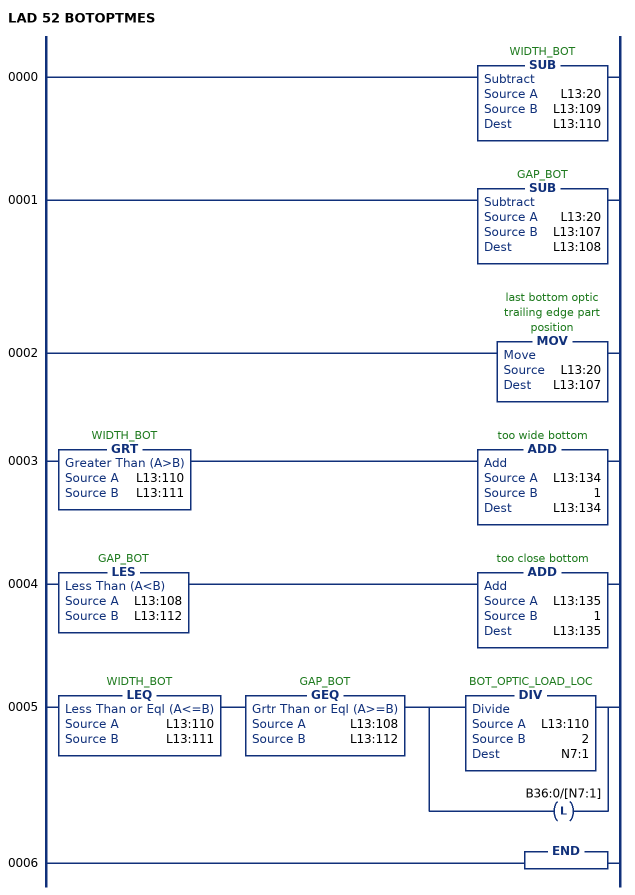
% Rung: 0 %
SOR SUB L13:20 L13:109 L13:110 EOR
%   L13:20  BOT_POSITION %
%   L13:109  BOT_LEAD_EDGE  "last bottom optic leading edge position" %
%   L13:110  WIDTH_BOT %
% Rung: 1 %
SOR SUB L13:20 L13:107 L13:108 EOR
%   L13:20  BOT_POSITION %
%   L13:107  "last bottom optic trailing edge part position" %
%   L13:108  GAP_BOT %
% Rung: 2 %
SOR MOV L13:20 L13:107 EOR
%   L13:20  BOT_POSITION %
%   L13:107  "last bottom optic trailing edge part position" %
% Rung: 3 %
SOR GRT L13:110 L13:111 ADD L13:134 1 L13:134 EOR
%   L13:110  WIDTH_BOT %
%   L13:111  BOT_MAX_WIDTH %
%   L13:134  "too wide bottom" %
% Rung: 4 %
SOR LES L13:108 L13:112 ADD L13:135 1 L13:135 EOR
%   L13:108  GAP_BOT %
%   L13:112  BOT_MIN_GAP %
%   L13:135  "too close bottom" %
% Rung: 5 %
SOR LEQ L13:110 L13:111 GEQ L13:108 L13:112 BST DIV L13:110 2 N7:1 NXB OTL B36:0/[N7:1] BND EOR
%   L13:110  WIDTH_BOT %
%   L13:111  BOT_MAX_WIDTH %
%   L13:108  GAP_BOT %
%   L13:112  BOT_MIN_GAP %
%   N7:1  BOT_OPTIC_LOAD_LOC %
%   B36:0  BOT_GOOD %
% Rung: 6 %
SOR END EOR

LADDER 60 "1 INS1"
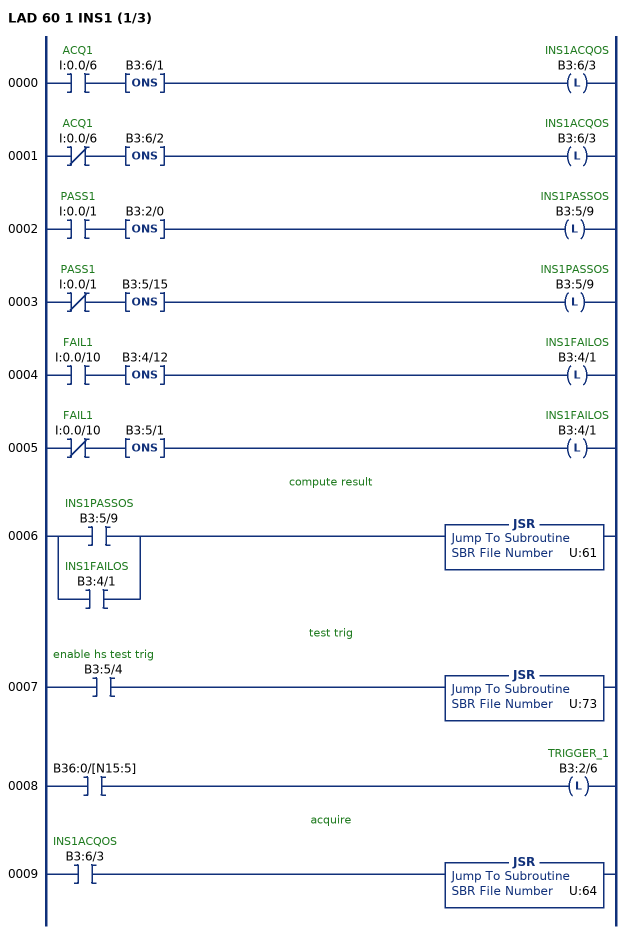
% Rung: 0 %
SOR XIC I:0.0/6 ONS B3:6/1 OTL B3:6/3 EOR
%   I:0.0/6  ACQ1 %
%   B3:6/3  INS1ACQOS %
% Rung: 1 %
SOR XIO I:0.0/6 ONS B3:6/2 OTL B3:6/3 EOR
%   I:0.0/6  ACQ1 %
%   B3:6/3  INS1ACQOS %
% Rung: 2 %
SOR XIC I:0.0/1 ONS B3:2/0 OTL B3:5/9 EOR
%   I:0.0/1  PASS1 %
%   B3:5/9  INS1PASSOS %
% Rung: 3 %
SOR XIO I:0.0/1 ONS B3:5/15 OTL B3:5/9 EOR
%   I:0.0/1  PASS1 %
%   B3:5/9  INS1PASSOS %
% Rung: 4 %
SOR XIC I:0.0/10 ONS B3:4/12 OTL B3:4/1 EOR
%   I:0.0/10  FAIL1 %
%   B3:4/1  INS1FAILOS %
% Rung: 5 %
SOR XIO I:0.0/10 ONS B3:5/1 OTL B3:4/1 EOR
%   I:0.0/10  FAIL1 %
%   B3:4/1  INS1FAILOS %
% Rung: 6 %
% compute result %
SOR BST XIC B3:5/9 NXB XIC B3:4/1 BND JSR U:61 EOR
%   B3:5/9  INS1PASSOS %
%   B3:4/1  INS1FAILOS %
% Rung: 7 %
% test trig %
SOR XIC B3:5/4 JSR U:73 EOR
%   B3:5/4  "enable hs test trig" %
% Rung: 8 %
SOR XIC B36:0/[N15:5] OTL B3:2/6 EOR
%   B36:0  BOT_GOOD %
%   N15:5  INS_1_TRIG_LOC %
%   B3:2/6  TRIGGER_1 %
% Rung: 9 %
% acquire %
SOR XIC B3:6/3 JSR U:64 EOR
%   B3:6/3  INS1ACQOS %

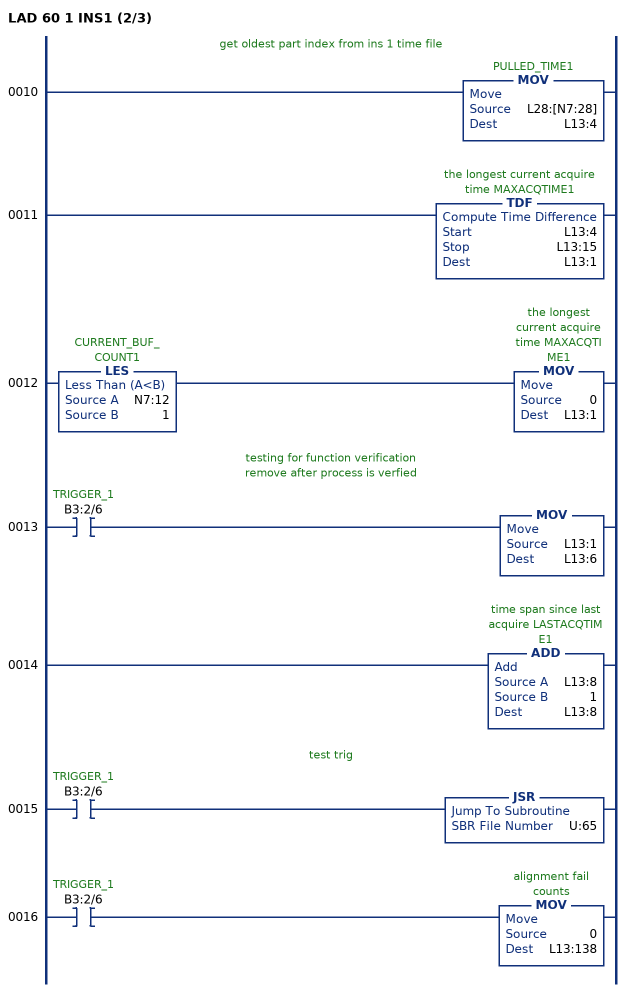
% Rung: 10 %
% get oldest part index from ins 1 time file %
SOR MOV L28:[N7:28] L13:4 EOR
%   N7:28  OLDEST_PART_INDEX1 %
%   L13:4  PULLED_TIME1 %
% Rung: 11 %
SOR TDF L13:4 L13:15 L13:1 EOR
%   L13:4  PULLED_TIME1 %
%   L13:15  THE_TIME %
%   L13:1  MAXACQTIME1  "the longest current acquire time" %
% Rung: 12 %
SOR LES N7:12 1 MOV 0 L13:1 EOR
%   N7:12  CURRENT_BUF_COUNT1 %
%   L13:1  MAXACQTIME1  "the longest current acquire time" %
% Rung: 13 %
% testing for function verification
% remove after process is verfied %
SOR XIC B3:2/6 MOV L13:1 L13:6 EOR
%   B3:2/6  TRIGGER_1 %
%   L13:1  MAXACQTIME1  "the longest current acquire time" %
% Rung: 14 %
SOR ADD L13:8 1 L13:8 EOR
%   L13:8  LASTACQTIME1  "time span since last acquire" %
% Rung: 15 %
% test trig %
SOR XIC B3:2/6 JSR U:65 EOR
%   B3:2/6  TRIGGER_1 %
% Rung: 16 %
SOR XIC B3:2/6 MOV 0 L13:138 EOR
%   B3:2/6  TRIGGER_1 %
%   L13:138  "alignment fail counts" %

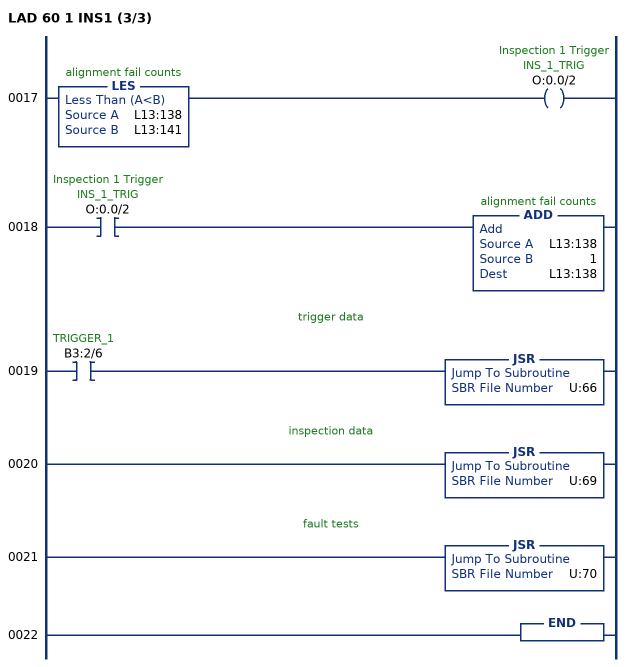
% Rung: 17 %
SOR LES L13:138 L13:141 OTE O:0.0/2 EOR
%   L13:138  "alignment fail counts" %
%   O:0.0/2  INS_1_TRIG  "Inspection 1 Trigger" %
% Rung: 18 %
SOR XIC O:0.0/2 ADD L13:138 1 L13:138 EOR
%   O:0.0/2  INS_1_TRIG  "Inspection 1 Trigger" %
%   L13:138  "alignment fail counts" %
% Rung: 19 %
% trigger data %
SOR XIC B3:2/6 JSR U:66 EOR
%   B3:2/6  TRIGGER_1 %
% Rung: 20 %
% inspection data %
SOR JSR U:69 EOR
% Rung: 21 %
% fault tests %
SOR JSR U:70 EOR
% Rung: 22 %
SOR END EOR

LADDER 61 "2 INS1RESU"
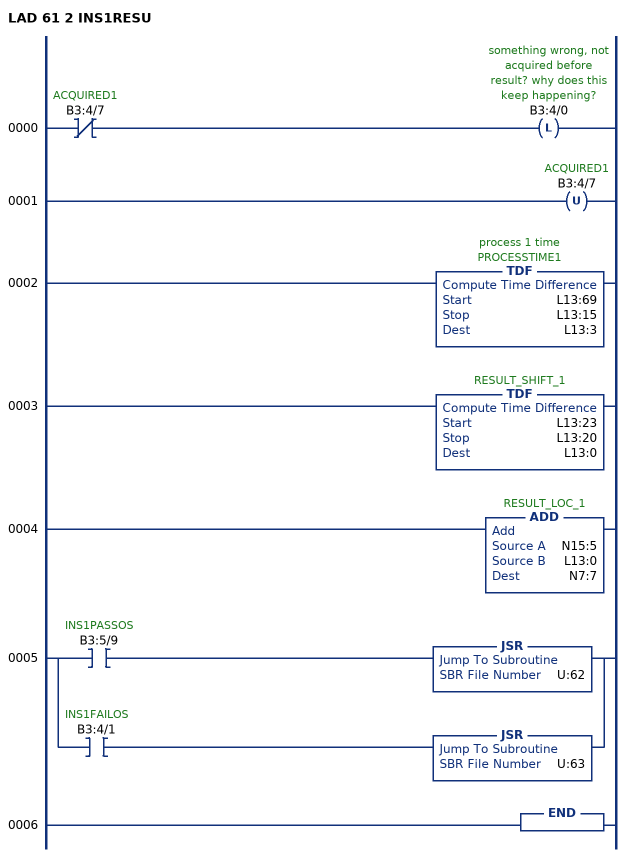
% Rung: 0 %
SOR XIO B3:4/7 OTL B3:4/0 EOR
%   B3:4/7  ACQUIRED1 %
%   B3:4/0  "something wrong, not acquired before result? why does this keep happening?" %
% Rung: 1 %
SOR OTU B3:4/7 EOR
%   B3:4/7  ACQUIRED1 %
% Rung: 2 %
SOR TDF L13:69 L13:15 L13:3 EOR
%   L13:69  TIMEOFACQ1  "the time of the last acquire" %
%   L13:15  THE_TIME %
%   L13:3  PROCESSTIME1  "process 1 time" %
% Rung: 3 %
SOR TDF L13:23 L13:20 L13:0 EOR
%   L13:23  PROCESS_START_POS_1 %
%   L13:20  BOT_POSITION %
%   L13:0  RESULT_SHIFT_1 %
% Rung: 4 %
SOR ADD N15:5 L13:0 N7:7 EOR
%   N15:5  INS_1_TRIG_LOC %
%   L13:0  RESULT_SHIFT_1 %
%   N7:7  RESULT_LOC_1 %
% Rung: 5 %
SOR BST XIC B3:5/9 JSR U:62 NXB XIC B3:4/1 JSR U:63 BND EOR
%   B3:5/9  INS1PASSOS %
%   B3:4/1  INS1FAILOS %
% Rung: 6 %
SOR END EOR

LADDER 62 "3 INS1PASS"
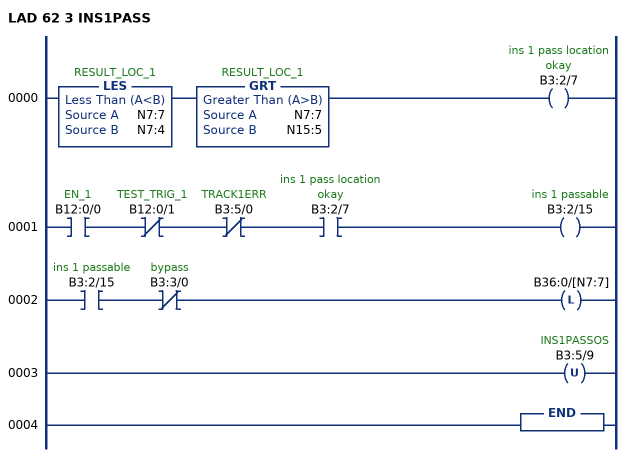
% Rung: 0 %
SOR LES N7:7 N7:4 GRT N7:7 N15:5 OTE B3:2/7 EOR
%   N7:7  RESULT_LOC_1 %
%   N7:4  INS1_MAX_SHIFT  "ins 1 maximum result location" %
%   N15:5  INS_1_TRIG_LOC %
%   B3:2/7  "ins 1 pass location okay" %
% Rung: 1 %
SOR XIC B12:0/0 XIO B12:0/1 XIO B3:5/0 XIC B3:2/7 OTE B3:2/15 EOR
%   B12:0/0  EN_1 %
%   B12:0/1  TEST_TRIG_1 %
%   B3:5/0  TRACK1ERR %
%   B3:2/7  "ins 1 pass location okay" %
%   B3:2/15  "ins 1 passable" %
% Rung: 2 %
SOR XIC B3:2/15 XIO B3:3/0 OTL B36:0/[N7:7] EOR
%   B3:2/15  "ins 1 passable" %
%   B3:3/0  "bypass" %
%   B36:0  BOT_GOOD %
%   N7:7  RESULT_LOC_1 %
% Rung: 3 %
SOR OTU B3:5/9 EOR
%   B3:5/9  INS1PASSOS %
% Rung: 4 %
SOR END EOR

LADDER 63 "4 INS1FAIL"
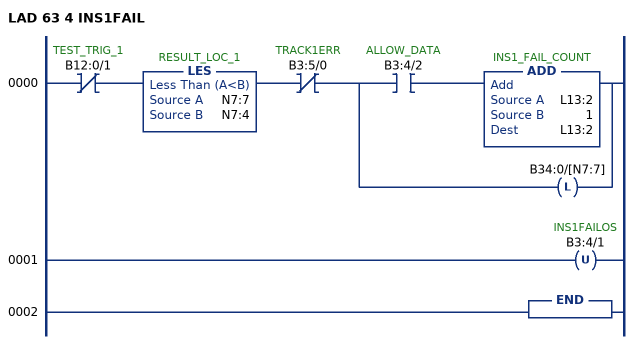
% Rung: 0 %
SOR XIO B12:0/1 LES N7:7 N7:4 XIO B3:5/0 BST XIC B3:4/2 ADD L13:2 1 L13:2 NXB OTL B34:0/[N7:7] BND EOR
%   B12:0/1  TEST_TRIG_1 %
%   N7:7  RESULT_LOC_1 %
%   N7:4  INS1_MAX_SHIFT  "ins 1 maximum result location" %
%   B3:5/0  TRACK1ERR %
%   B3:4/2  ALLOW_DATA %
%   L13:2  INS1_FAIL_COUNT %
%   B34:0  BOT_NG %
% Rung: 1 %
SOR OTU B3:4/1 EOR
%   B3:4/1  INS1FAILOS %
% Rung: 2 %
SOR END EOR

LADDER 64 "5 INS1ACQ"
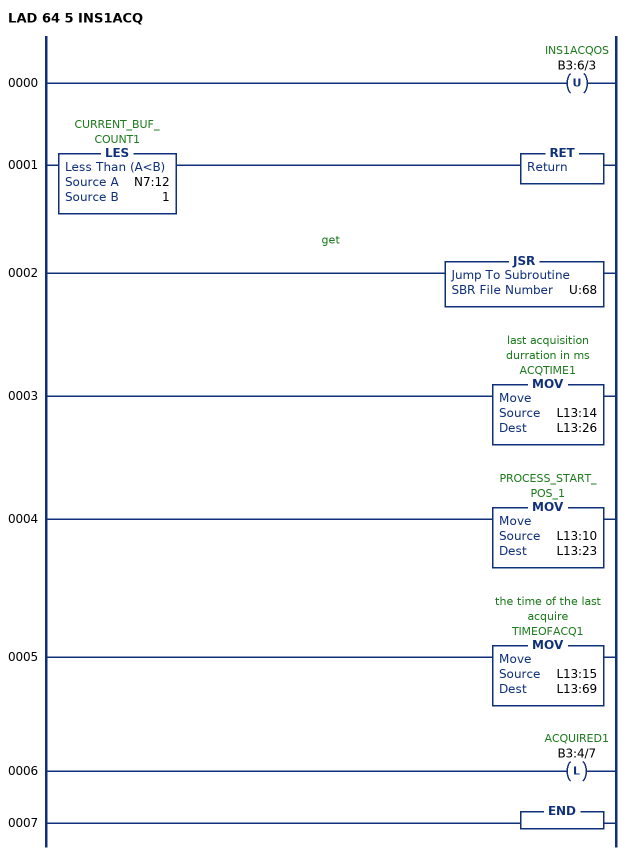
% Rung: 0 %
SOR OTU B3:6/3 EOR
%   B3:6/3  INS1ACQOS %
% Rung: 1 %
SOR LES N7:12 1 RET EOR
%   N7:12  CURRENT_BUF_COUNT1 %
% Rung: 2 %
% get %
SOR JSR U:68 EOR
% Rung: 3 %
SOR MOV L13:14 L13:26 EOR
%   L13:14  TIME_SPAN1 %
%   L13:26  ACQTIME1  "last acquisition durration in ms" %
% Rung: 4 %
SOR MOV L13:10 L13:23 EOR
%   L13:10  PULLED_POSITION1 %
%   L13:23  PROCESS_START_POS_1 %
% Rung: 5 %
SOR MOV L13:15 L13:69 EOR
%   L13:15  THE_TIME %
%   L13:69  TIMEOFACQ1  "the time of the last acquire" %
% Rung: 6 %
SOR OTL B3:4/7 EOR
%   B3:4/7  ACQUIRED1 %
% Rung: 7 %
SOR END EOR

LADDER 65 "6 Q1TESTTR"
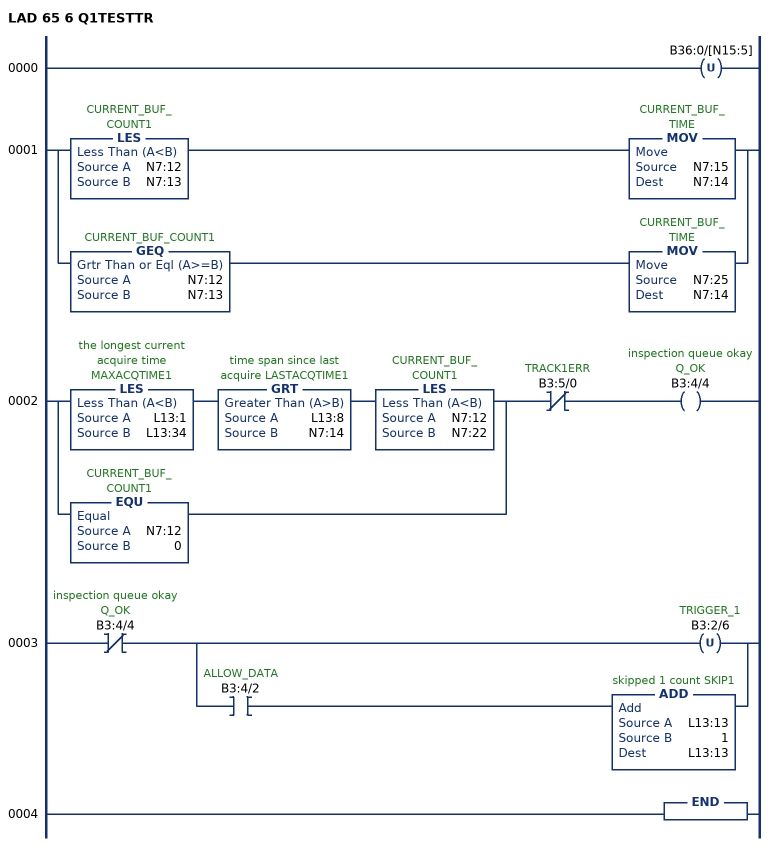
% Rung: 0 %
SOR OTU B36:0/[N15:5] EOR
%   B36:0  BOT_GOOD %
%   N15:5  INS_1_TRIG_LOC %
% Rung: 1 %
SOR BST LES N7:12 N7:13 MOV N7:15 N7:14 NXB GEQ N7:12 N7:13 MOV N7:25 N7:14 BND EOR
%   N7:12  CURRENT_BUF_COUNT1 %
%   N7:13  BUF_TRANS  "cam to pc buf transition" %
%   N7:15  CAM_BUF_TIME  "cam buf time" %
%   N7:14  CURRENT_BUF_TIME %
%   N7:25  PC_BUF_TIME  "pc buf time" %
% Rung: 2 %
SOR BST LES L13:1 L13:34 GRT L13:8 N7:14 LES N7:12 N7:22 NXB EQU N7:12 0 BND XIO B3:5/0 OTE B3:4/4 EOR
%   L13:1  MAXACQTIME1  "the longest current acquire time" %
%   L13:34  MAX_ACQ_ALL  "absolute max acquire time before bypass trigger" %
%   L13:8  LASTACQTIME1  "time span since last acquire" %
%   N7:14  CURRENT_BUF_TIME %
%   N7:12  CURRENT_BUF_COUNT1 %
%   N7:22  MAX_BUF_ALL  "max buffer count alowed before bypass" %
%   B3:5/0  TRACK1ERR %
%   B3:4/4  Q_OK  "inspection queue okay" %
% Rung: 3 %
SOR XIO B3:4/4 BST OTU B3:2/6 NXB XIC B3:4/2 ADD L13:13 1 L13:13 BND EOR
%   B3:4/4  Q_OK  "inspection queue okay" %
%   B3:2/6  TRIGGER_1 %
%   B3:4/2  ALLOW_DATA %
%   L13:13  SKIP1  "skipped 1 count" %
% Rung: 4 %
SOR END EOR

LADDER 66 "7 INS1TRIG"
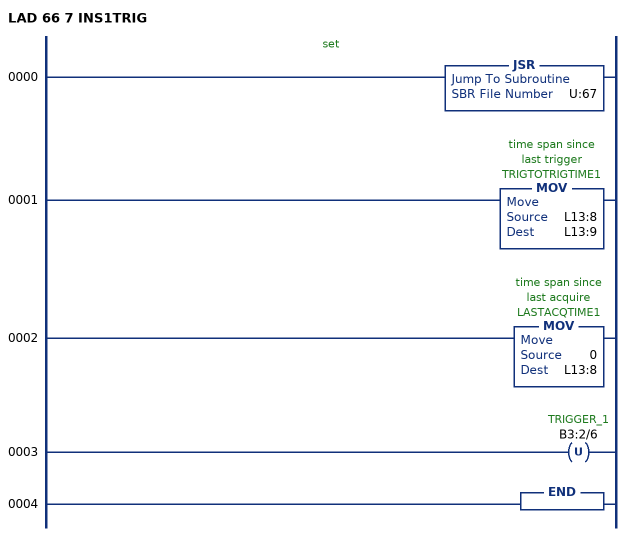
% Rung: 0 %
% set %
SOR JSR U:67 EOR
% Rung: 1 %
SOR MOV L13:8 L13:9 EOR
%   L13:8  LASTACQTIME1  "time span since last acquire" %
%   L13:9  TRIGTOTRIGTIME1  "time span since last trigger" %
% Rung: 2 %
SOR MOV 0 L13:8 EOR
%   L13:8  LASTACQTIME1  "time span since last acquire" %
% Rung: 3 %
SOR OTU B3:2/6 EOR
%   B3:2/6  TRIGGER_1 %
% Rung: 4 %
SOR END EOR

LADDER 67 "8 FIFO1SET"
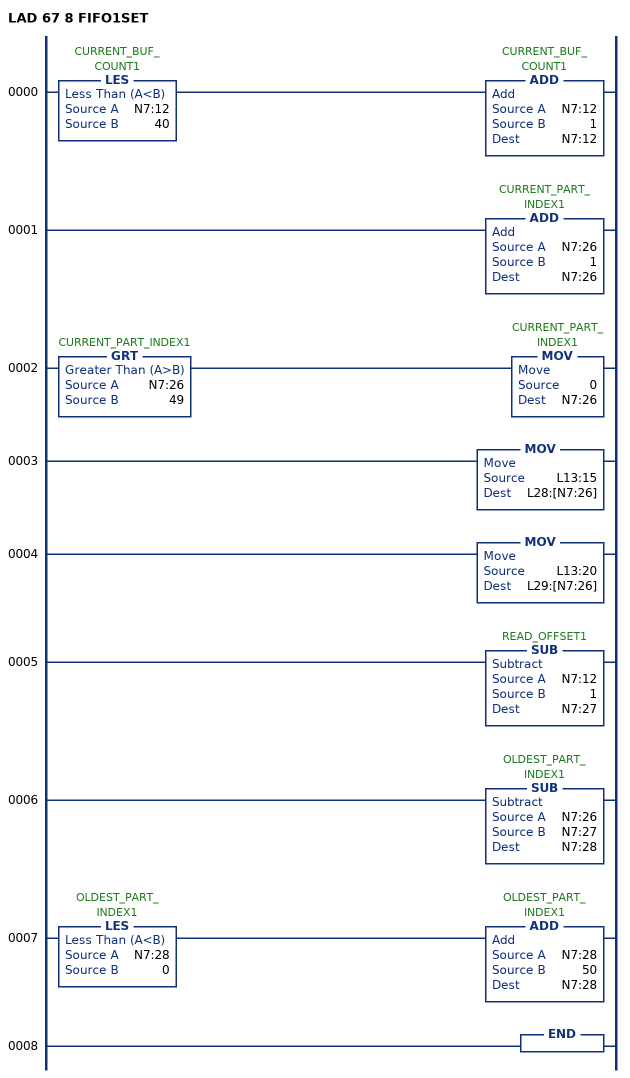
% Rung: 0 %
SOR LES N7:12 40 ADD N7:12 1 N7:12 EOR
%   N7:12  CURRENT_BUF_COUNT1 %
% Rung: 1 %
SOR ADD N7:26 1 N7:26 EOR
%   N7:26  CURRENT_PART_INDEX1 %
% Rung: 2 %
SOR GRT N7:26 49 MOV 0 N7:26 EOR
%   N7:26  CURRENT_PART_INDEX1 %
% Rung: 3 %
SOR MOV L13:15 L28:[N7:26] EOR
%   L13:15  THE_TIME %
%   N7:26  CURRENT_PART_INDEX1 %
% Rung: 4 %
SOR MOV L13:20 L29:[N7:26] EOR
%   L13:20  BOT_POSITION %
%   N7:26  CURRENT_PART_INDEX1 %
% Rung: 5 %
SOR SUB N7:12 1 N7:27 EOR
%   N7:12  CURRENT_BUF_COUNT1 %
%   N7:27  READ_OFFSET1 %
% Rung: 6 %
SOR SUB N7:26 N7:27 N7:28 EOR
%   N7:26  CURRENT_PART_INDEX1 %
%   N7:27  READ_OFFSET1 %
%   N7:28  OLDEST_PART_INDEX1 %
% Rung: 7 %
SOR LES N7:28 0 ADD N7:28 50 N7:28 EOR
%   N7:28  OLDEST_PART_INDEX1 %
% Rung: 8 %
SOR END EOR

LADDER 68 "9 FIFO1GET"
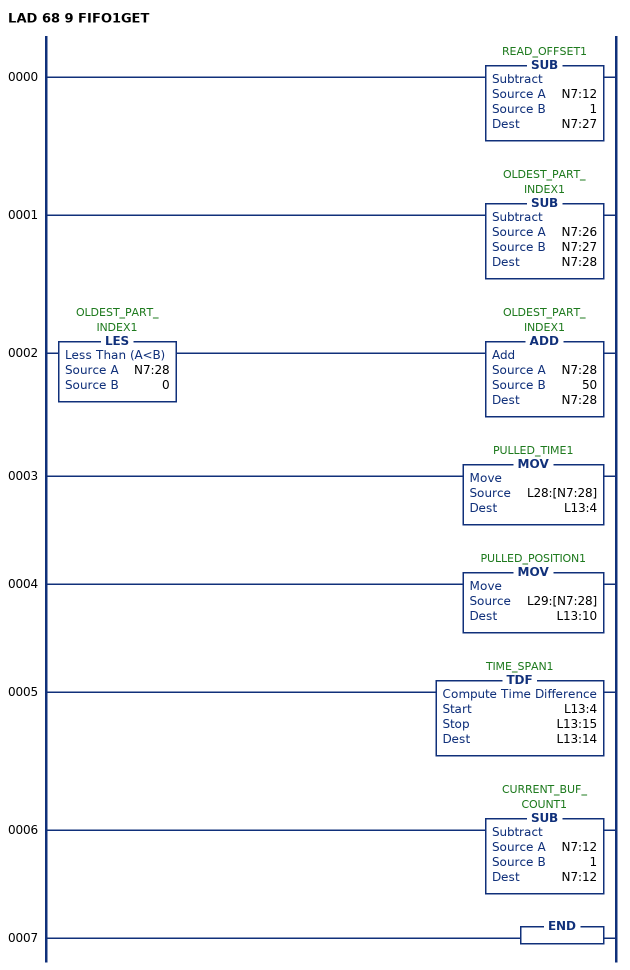
% Rung: 0 %
SOR SUB N7:12 1 N7:27 EOR
%   N7:12  CURRENT_BUF_COUNT1 %
%   N7:27  READ_OFFSET1 %
% Rung: 1 %
SOR SUB N7:26 N7:27 N7:28 EOR
%   N7:26  CURRENT_PART_INDEX1 %
%   N7:27  READ_OFFSET1 %
%   N7:28  OLDEST_PART_INDEX1 %
% Rung: 2 %
SOR LES N7:28 0 ADD N7:28 50 N7:28 EOR
%   N7:28  OLDEST_PART_INDEX1 %
% Rung: 3 %
SOR MOV L28:[N7:28] L13:4 EOR
%   N7:28  OLDEST_PART_INDEX1 %
%   L13:4  PULLED_TIME1 %
% Rung: 4 %
SOR MOV L29:[N7:28] L13:10 EOR
%   N7:28  OLDEST_PART_INDEX1 %
%   L13:10  PULLED_POSITION1 %
% Rung: 5 %
SOR TDF L13:4 L13:15 L13:14 EOR
%   L13:4  PULLED_TIME1 %
%   L13:15  THE_TIME %
%   L13:14  TIME_SPAN1 %
% Rung: 6 %
SOR SUB N7:12 1 N7:12 EOR
%   N7:12  CURRENT_BUF_COUNT1 %
% Rung: 7 %
SOR END EOR

LADDER 69 "10INSDATA1"
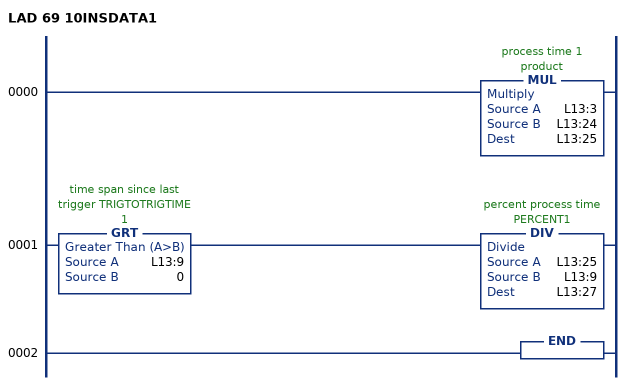
% Rung: 0 %
SOR MUL L13:3 L13:24 L13:25 EOR
%   L13:3  PROCESSTIME1  "process 1 time" %
%   L13:24  "multiplyer to make devision come out to a percentage" %
%   L13:25  "process time 1 product" %
% Rung: 1 %
SOR GRT L13:9 0 DIV L13:25 L13:9 L13:27 EOR
%   L13:9  TRIGTOTRIGTIME1  "time span since last trigger" %
%   L13:25  "process time 1 product" %
%   L13:27  PERCENT1  "percent process time" %
% Rung: 2 %
SOR END EOR

LADDER 70 "11TSTFALT1"
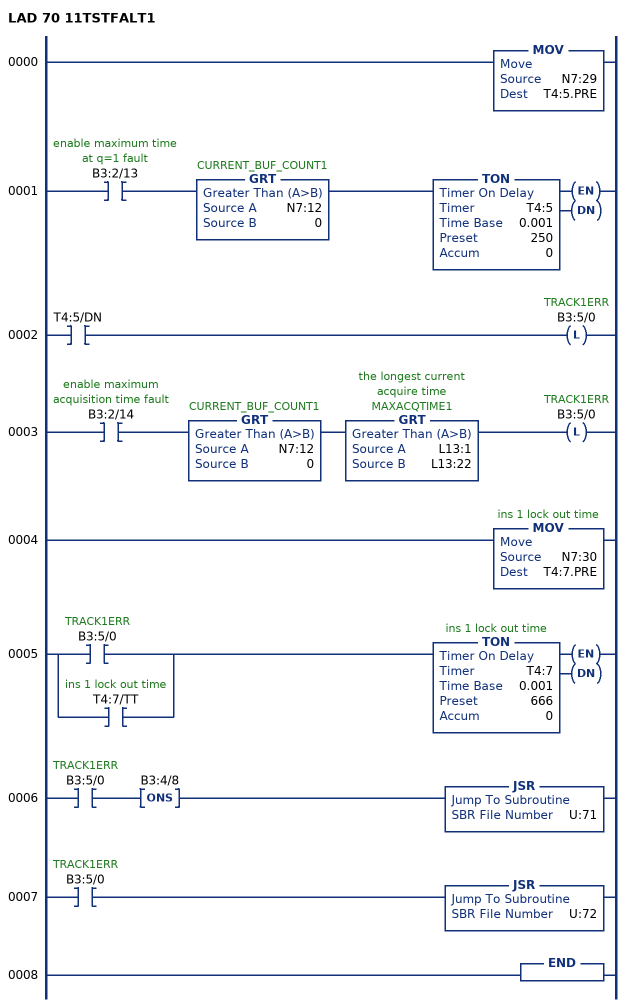
% Rung: 0 %
SOR MOV N7:29 T4:5.PRE EOR
%   N7:29  "max allowed ms time for q to be above 1 if safe fault is used" %
% Rung: 1 %
SOR XIC B3:2/13 GRT N7:12 0 TON T4:5 0.001 250 0 EOR
%   B3:2/13  "enable maximum time at q=1 fault" %
%   N7:12  CURRENT_BUF_COUNT1 %
% Rung: 2 %
SOR XIC T4:5/DN OTL B3:5/0 EOR
%   B3:5/0  TRACK1ERR %
% Rung: 3 %
SOR XIC B3:2/14 GRT N7:12 0 GRT L13:1 L13:22 OTL B3:5/0 EOR
%   B3:2/14  "enable maximum acquisition time fault" %
%   N7:12  CURRENT_BUF_COUNT1 %
%   L13:1  MAXACQTIME1  "the longest current acquire time" %
%   L13:22  "maximum of the longest acquire time allowed if maximum acquire time fault is enabled" %
%   B3:5/0  TRACK1ERR %
% Rung: 4 %
SOR MOV N7:30 T4:7.PRE EOR
%   N7:30  "ms time setting to lock out inspection to give all pending images a chance to clear" %
%   T4:7  "ins 1 lock out time" %
% Rung: 5 %
SOR BST XIC B3:5/0 NXB XIC T4:7/TT BND TON T4:7 0.001 666 0 EOR
%   B3:5/0  TRACK1ERR %
%   T4:7  "ins 1 lock out time" %
% Rung: 6 %
SOR XIC B3:5/0 ONS B3:4/8 JSR U:71 EOR
%   B3:5/0  TRACK1ERR %
% Rung: 7 %
SOR XIC B3:5/0 JSR U:72 EOR
%   B3:5/0  TRACK1ERR %
% Rung: 8 %
SOR END EOR

LADDER 71 "12INS1FIX1"
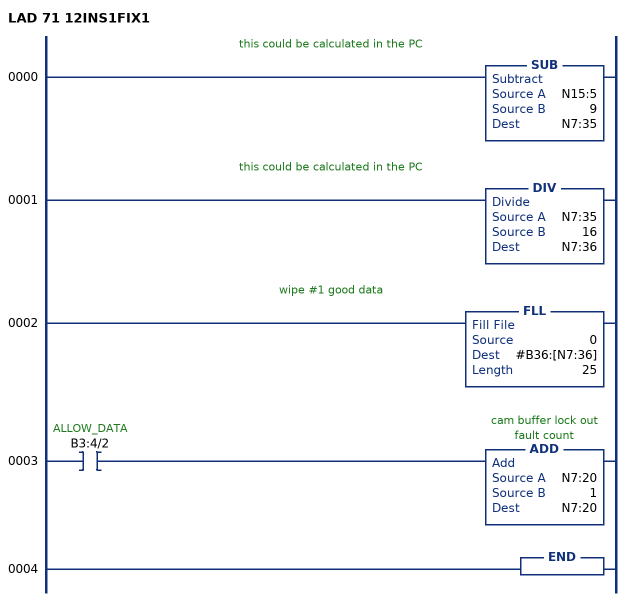
% Rung: 0 %
% this could be calculated in the PC %
SOR SUB N15:5 9 N7:35 EOR
%   N15:5  INS_1_TRIG_LOC %
% Rung: 1 %
% this could be calculated in the PC %
SOR DIV N7:35 16 N7:36 EOR
% Rung: 2 %
% wipe #1 good data %
SOR FLL 0 #B36:[N7:36] 25 EOR
% Rung: 3 %
SOR XIC B3:4/2 ADD N7:20 1 N7:20 EOR
%   B3:4/2  ALLOW_DATA %
%   N7:20  "cam buffer lock out fault count" %
% Rung: 4 %
SOR END EOR

LADDER 72 "13INS1FIX2"
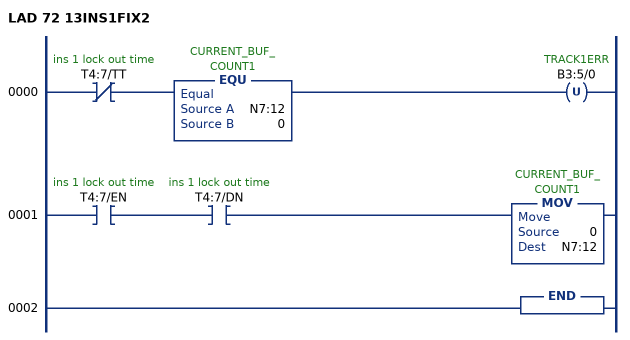
% Rung: 0 %
SOR XIO T4:7/TT EQU N7:12 0 OTU B3:5/0 EOR
%   T4:7  "ins 1 lock out time" %
%   N7:12  CURRENT_BUF_COUNT1 %
%   B3:5/0  TRACK1ERR %
% Rung: 1 %
SOR XIC T4:7/EN XIC T4:7/DN MOV 0 N7:12 EOR
%   T4:7  "ins 1 lock out time" %
%   N7:12  CURRENT_BUF_COUNT1 %
% Rung: 2 %
SOR END EOR

LADDER 73 "14 HSTRIG1"
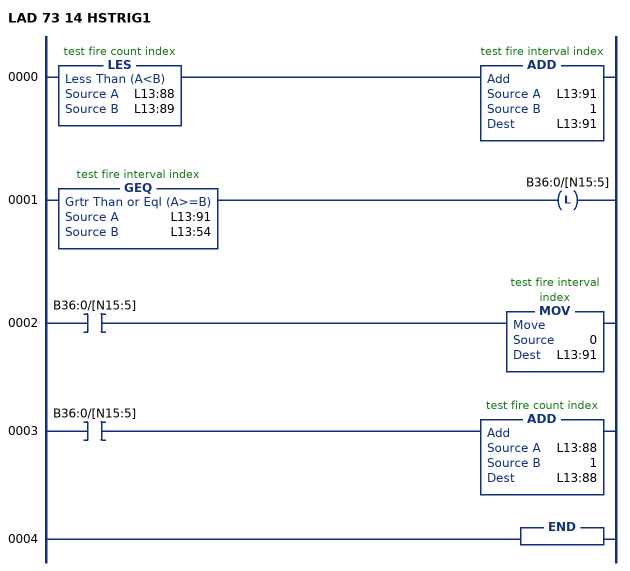
% Rung: 0 %
SOR LES L13:88 L13:89 ADD L13:91 1 L13:91 EOR
%   L13:88  "test fire count index" %
%   L13:89  "test fire count" %
%   L13:91  "test fire interval index" %
% Rung: 1 %
SOR GEQ L13:91 L13:54 OTL B36:0/[N15:5] EOR
%   L13:91  "test fire interval index" %
%   L13:54  "test fire interval" %
%   B36:0  BOT_GOOD %
%   N15:5  INS_1_TRIG_LOC %
% Rung: 2 %
SOR XIC B36:0/[N15:5] MOV 0 L13:91 EOR
%   B36:0  BOT_GOOD %
%   N15:5  INS_1_TRIG_LOC %
%   L13:91  "test fire interval index" %
% Rung: 3 %
SOR XIC B36:0/[N15:5] ADD L13:88 1 L13:88 EOR
%   B36:0  BOT_GOOD %
%   N15:5  INS_1_TRIG_LOC %
%   L13:88  "test fire count index" %
% Rung: 4 %
SOR END EOR

LADDER 80 "XFER"
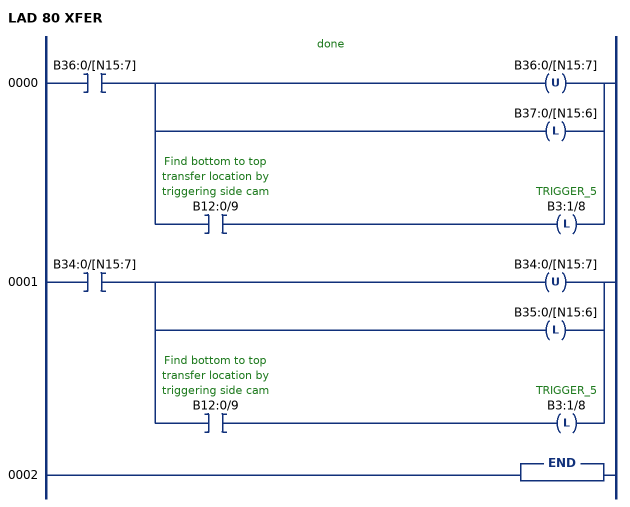
% Rung: 0 %
% done %
SOR XIC B36:0/[N15:7] BST OTU B36:0/[N15:7] NXB OTL B37:0/[N15:6] NXB XIC B12:0/9 OTL B3:1/8 BND EOR
%   B36:0  BOT_GOOD %
%   N15:7  XFER_OUT_LOC %
%   N15:6  XFER_IN_LOC %
%   B12:0/9  "Find bottom to top transfer location by triggering side cam" %
%   B3:1/8  TRIGGER_5 %
% Rung: 1 %
SOR XIC B34:0/[N15:7] BST OTU B34:0/[N15:7] NXB OTL B35:0/[N15:6] NXB XIC B12:0/9 OTL B3:1/8 BND EOR
%   B34:0  BOT_NG %
%   N15:7  XFER_OUT_LOC %
%   B35:0  TOP_NG %
%   N15:6  XFER_IN_LOC %
%   B12:0/9  "Find bottom to top transfer location by triggering side cam" %
%   B3:1/8  TRIGGER_5 %
% Rung: 2 %
SOR END EOR

LADDER 90 "TOPOPTIC"
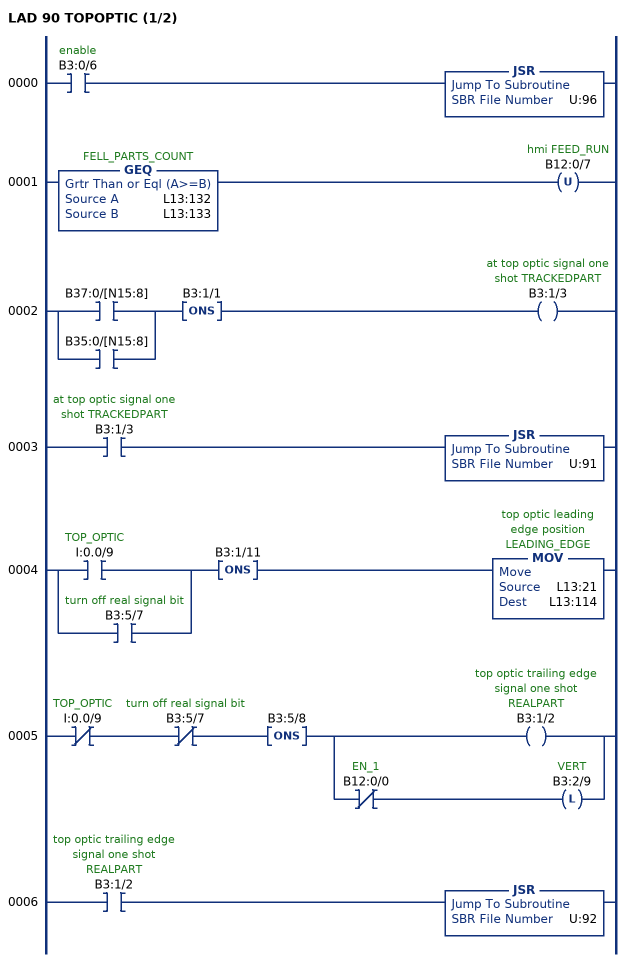
% Rung: 0 %
SOR XIC B3:0/6 JSR U:96 EOR
%   B3:0/6  "enable" %
% Rung: 1 %
SOR GEQ L13:132 L13:133 OTU B12:0/7 EOR
%   L13:132  FELL_PARTS_COUNT %
%   L13:133  FELL_PARTS_LIMIT %
%   B12:0/7  FEED_RUN  "hmi" %
% Rung: 2 %
SOR BST XIC B37:0/[N15:8] NXB XIC B35:0/[N15:8] BND ONS B3:1/1 OTE B3:1/3 EOR
%   N15:8  TOP_OPTIC_LOC %
%   B35:0  TOP_NG %
%   B3:1/3  TRACKEDPART  "at top optic signal one shot" %
% Rung: 3 %
SOR XIC B3:1/3 JSR U:91 EOR
%   B3:1/3  TRACKEDPART  "at top optic signal one shot" %
% Rung: 4 %
SOR BST XIC I:0.0/9 NXB XIC B3:5/7 BND ONS B3:1/11 MOV L13:21 L13:114 EOR
%   I:0.0/9  TOP_OPTIC %
%   B3:5/7  "turn off real signal bit" %
%   L13:21  TOP_POSITION %
%   L13:114  LEADING_EDGE  "top optic leading edge position" %
% Rung: 5 %
SOR XIO I:0.0/9 XIO B3:5/7 ONS B3:5/8 BST OTE B3:1/2 NXB XIO B12:0/0 OTL B3:2/9 BND EOR
%   I:0.0/9  TOP_OPTIC %
%   B3:5/7  "turn off real signal bit" %
%   B3:1/2  REALPART  "top optic trailing edge signal one shot" %
%   B12:0/0  EN_1 %
%   B3:2/9  VERT %
% Rung: 6 %
SOR XIC B3:1/2 JSR U:92 EOR
%   B3:1/2  REALPART  "top optic trailing edge signal one shot" %

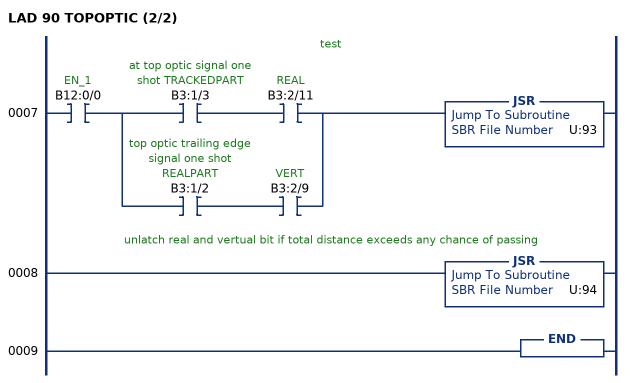
% Rung: 7 %
% test %
SOR XIC B12:0/0 BST XIC B3:1/3 XIC B3:2/11 NXB XIC B3:1/2 XIC B3:2/9 BND JSR U:93 EOR
%   B12:0/0  EN_1 %
%   B3:1/3  TRACKEDPART  "at top optic signal one shot" %
%   B3:2/11  REAL %
%   B3:1/2  REALPART  "top optic trailing edge signal one shot" %
%   B3:2/9  VERT %
% Rung: 8 %
% unlatch real and vertual bit if total distance exceeds any chance of passing %
SOR JSR U:94 EOR
% Rung: 9 %
SOR END EOR

LADDER 91 "TOPOPVERT"
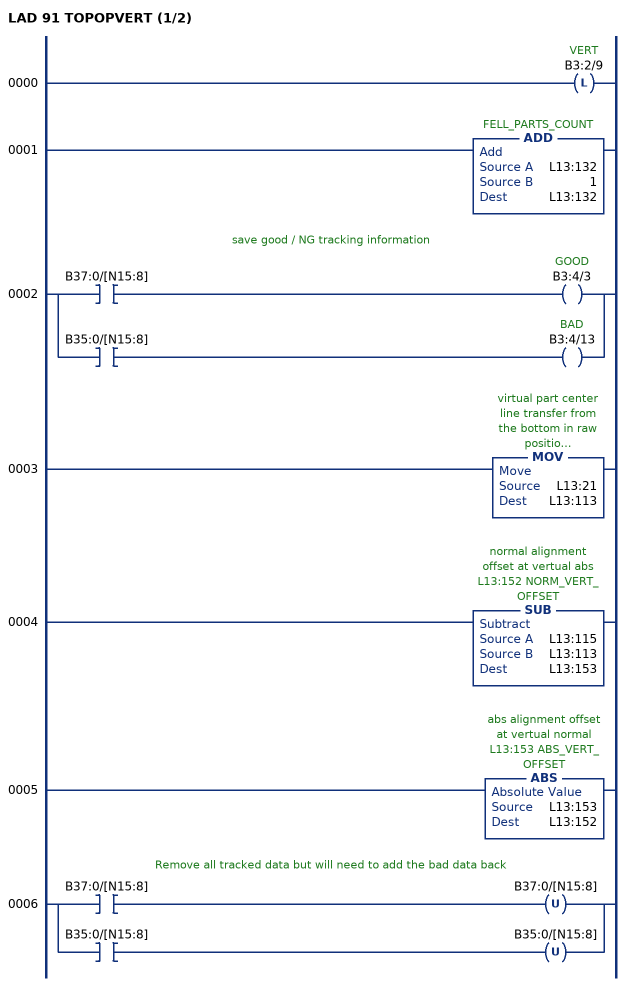
% Rung: 0 %
SOR OTL B3:2/9 EOR
%   B3:2/9  VERT %
% Rung: 1 %
SOR ADD L13:132 1 L13:132 EOR
%   L13:132  FELL_PARTS_COUNT %
% Rung: 2 %
% save good / NG tracking information %
SOR BST XIC B37:0/[N15:8] OTE B3:4/3 NXB XIC B35:0/[N15:8] OTE B3:4/13 BND EOR
%   N15:8  TOP_OPTIC_LOC %
%   B3:4/3  GOOD %
%   B35:0  TOP_NG %
%   B3:4/13  BAD %
% Rung: 3 %
SOR MOV L13:21 L13:113 EOR
%   L13:21  TOP_POSITION %
%   L13:113  VERTUAL_PT_RAW_CL  "virtual part center line transfer from the bottom in raw position" %
% Rung: 4 %
SOR SUB L13:115 L13:113 L13:153 EOR
%   L13:115  TRAILING_EDGE_RAW  "top optic trailing edge position" %
%   L13:113  VERTUAL_PT_RAW_CL  "virtual part center line transfer from the bottom in raw position" %
%   L13:153  NORM_VERT_OFFSET  "normal alignment offset at vertual abs L13:152" %
% Rung: 5 %
SOR ABS L13:153 L13:152 EOR
%   L13:153  NORM_VERT_OFFSET  "normal alignment offset at vertual abs L13:152" %
%   L13:152  ABS_VERT_OFFSET  "abs alignment offset at vertual normal L13:153" %
% Rung: 6 %
% Remove all tracked data but will need to add the bad data back %
SOR BST XIC B37:0/[N15:8] OTU B37:0/[N15:8] NXB XIC B35:0/[N15:8] OTU B35:0/[N15:8] BND EOR
%   N15:8  TOP_OPTIC_LOC %
%   B35:0  TOP_NG %

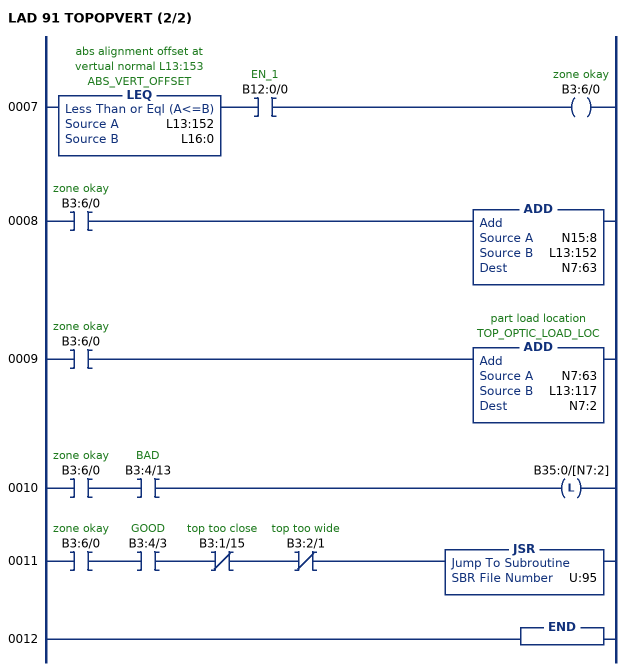
% Rung: 7 %
SOR LEQ L13:152 L16:0 XIC B12:0/0 OTE B3:6/0 EOR
%   L13:152  ABS_VERT_OFFSET  "abs alignment offset at vertual normal L13:153" %
%   L16:0  MAX_OFFSET %
%   B12:0/0  EN_1 %
%   B3:6/0  "zone okay" %
% Rung: 8 %
SOR XIC B3:6/0 ADD N15:8 L13:152 N7:63 EOR
%   B3:6/0  "zone okay" %
%   N15:8  TOP_OPTIC_LOC %
%   L13:152  ABS_VERT_OFFSET  "abs alignment offset at vertual normal L13:153" %
% Rung: 9 %
SOR XIC B3:6/0 ADD N7:63 L13:117 N7:2 EOR
%   B3:6/0  "zone okay" %
%   L13:117  HALF_WIDTH  "1/2 width top" %
%   N7:2  TOP_OPTIC_LOAD_LOC  "part load location" %
% Rung: 10 %
SOR XIC B3:6/0 XIC B3:4/13 OTL B35:0/[N7:2] EOR
%   B3:6/0  "zone okay" %
%   B3:4/13  BAD %
%   B35:0  TOP_NG %
%   N7:2  TOP_OPTIC_LOAD_LOC  "part load location" %
% Rung: 11 %
SOR XIC B3:6/0 XIC B3:4/3 XIO B3:1/15 XIO B3:2/1 JSR U:95 EOR
%   B3:6/0  "zone okay" %
%   B3:4/3  GOOD %
%   B3:1/15  "top too close" %
%   B3:2/1  "top too wide" %
% Rung: 12 %
SOR END EOR

LADDER 92 "TOPOPREAL"
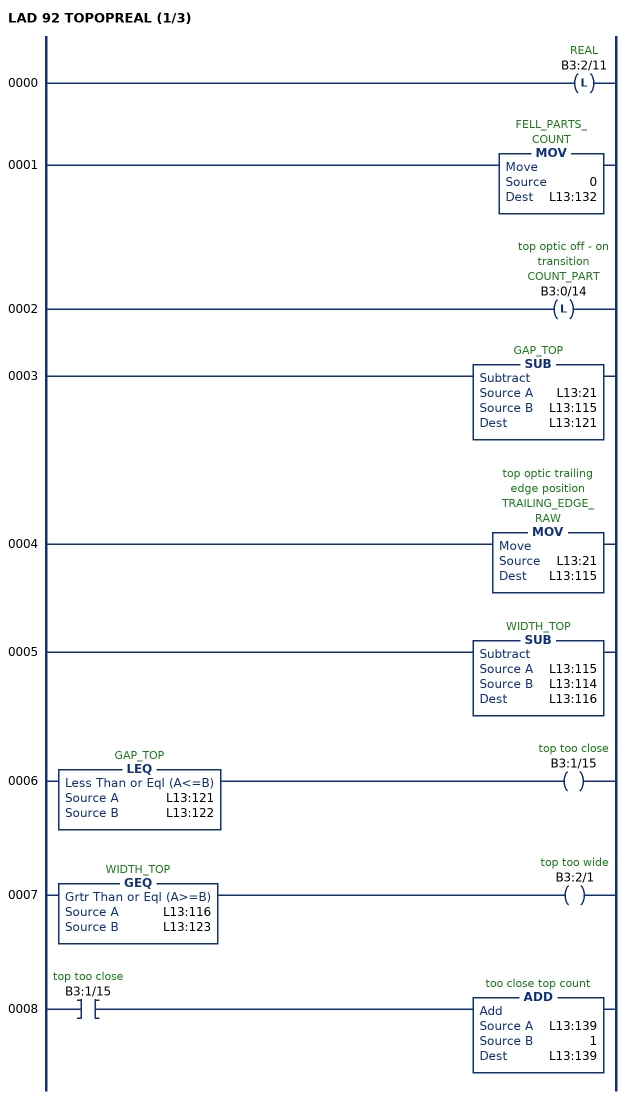
% Rung: 0 %
SOR OTL B3:2/11 EOR
%   B3:2/11  REAL %
% Rung: 1 %
SOR MOV 0 L13:132 EOR
%   L13:132  FELL_PARTS_COUNT %
% Rung: 2 %
SOR OTL B3:0/14 EOR
%   B3:0/14  COUNT_PART  "top optic off - on transition" %
% Rung: 3 %
SOR SUB L13:21 L13:115 L13:121 EOR
%   L13:21  TOP_POSITION %
%   L13:115  TRAILING_EDGE_RAW  "top optic trailing edge position" %
%   L13:121  GAP_TOP %
% Rung: 4 %
SOR MOV L13:21 L13:115 EOR
%   L13:21  TOP_POSITION %
%   L13:115  TRAILING_EDGE_RAW  "top optic trailing edge position" %
% Rung: 5 %
SOR SUB L13:115 L13:114 L13:116 EOR
%   L13:115  TRAILING_EDGE_RAW  "top optic trailing edge position" %
%   L13:114  LEADING_EDGE  "top optic leading edge position" %
%   L13:116  WIDTH_TOP %
% Rung: 6 %
SOR LEQ L13:121 L13:122 OTE B3:1/15 EOR
%   L13:121  GAP_TOP %
%   L13:122  MIN_GAP_TOP %
%   B3:1/15  "top too close" %
% Rung: 7 %
SOR GEQ L13:116 L13:123 OTE B3:2/1 EOR
%   L13:116  WIDTH_TOP %
%   L13:123  MAX_WIDTH_TOP %
%   B3:2/1  "top too wide" %
% Rung: 8 %
SOR XIC B3:1/15 ADD L13:139 1 L13:139 EOR
%   B3:1/15  "top too close" %
%   L13:139  "too close top count" %

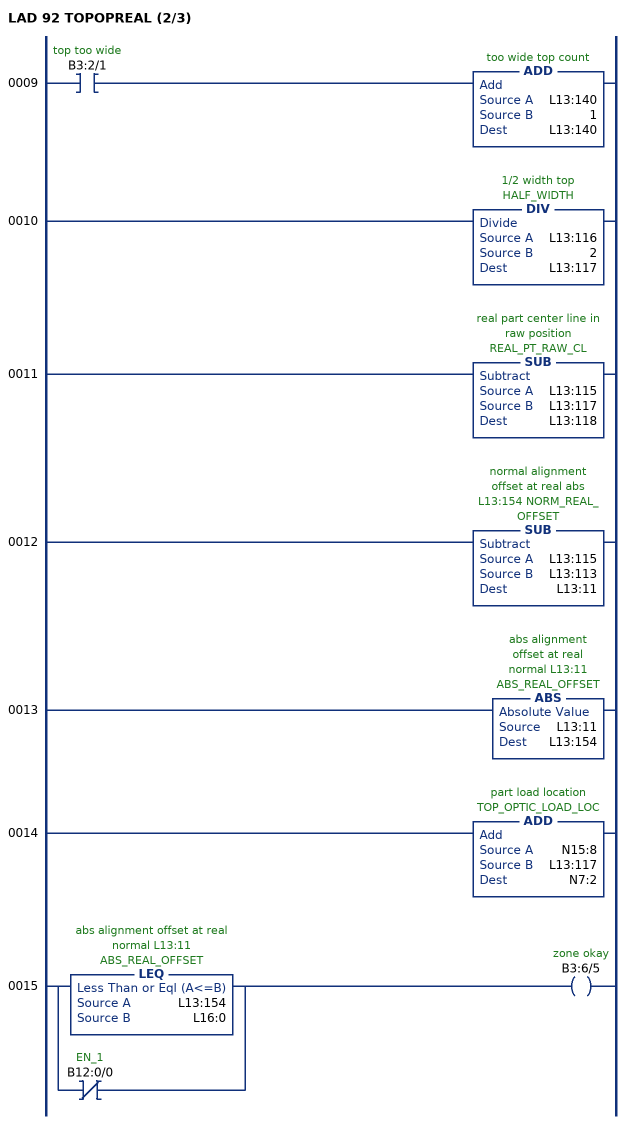
% Rung: 9 %
SOR XIC B3:2/1 ADD L13:140 1 L13:140 EOR
%   B3:2/1  "top too wide" %
%   L13:140  "too wide top count" %
% Rung: 10 %
SOR DIV L13:116 2 L13:117 EOR
%   L13:116  WIDTH_TOP %
%   L13:117  HALF_WIDTH  "1/2 width top" %
% Rung: 11 %
SOR SUB L13:115 L13:117 L13:118 EOR
%   L13:115  TRAILING_EDGE_RAW  "top optic trailing edge position" %
%   L13:117  HALF_WIDTH  "1/2 width top" %
%   L13:118  REAL_PT_RAW_CL  "real part center line in raw position" %
% Rung: 12 %
SOR SUB L13:115 L13:113 L13:11 EOR
%   L13:115  TRAILING_EDGE_RAW  "top optic trailing edge position" %
%   L13:113  VERTUAL_PT_RAW_CL  "virtual part center line transfer from the bottom in raw position" %
%   L13:11  NORM_REAL_OFFSET  "normal alignment offset at real abs L13:154" %
% Rung: 13 %
SOR ABS L13:11 L13:154 EOR
%   L13:11  NORM_REAL_OFFSET  "normal alignment offset at real abs L13:154" %
%   L13:154  ABS_REAL_OFFSET  "abs alignment offset at real normal L13:11" %
% Rung: 14 %
SOR ADD N15:8 L13:117 N7:2 EOR
%   N15:8  TOP_OPTIC_LOC %
%   L13:117  HALF_WIDTH  "1/2 width top" %
%   N7:2  TOP_OPTIC_LOAD_LOC  "part load location" %
% Rung: 15 %
SOR BST LEQ L13:154 L16:0 NXB XIO B12:0/0 BND OTE B3:6/5 EOR
%   L13:154  ABS_REAL_OFFSET  "abs alignment offset at real normal L13:11" %
%   L16:0  MAX_OFFSET %
%   B12:0/0  EN_1 %
%   B3:6/5  "zone okay" %

